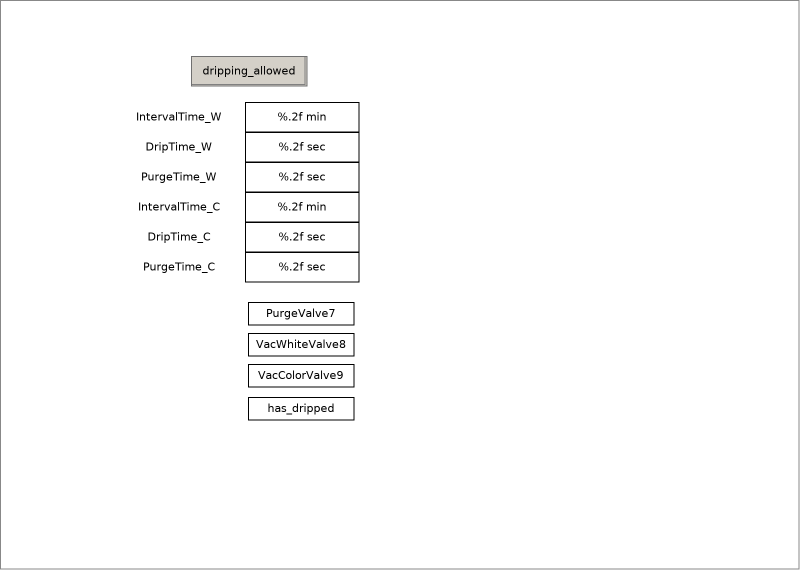
VISUALIZATION VIS_Drip_purge  // 800x570
    Button (191,56 116x30), "dripping_allowed", colour toggle: GVL_API.stMU.dripping_allowed
        toggle GVL_API.stMU.dripping_allowed
    RoundedRectangle (248,302 106x23), "PurgeValve7", colour toggle: P_MaintenanceUnit.FB_drip_purge.PurgeValve7
    Label (122,102 114x30), "IntervalTime_W"
    Label (122,132 114x30), "DripTime_W"
    Label (122,222 114x30), "DripTime_C"
    Label (122,162 114x30), "PurgeTime_W"
    Label (122,192 114x30), "IntervalTime_C"
    Label (122,252 114x30), "PurgeTime_C"
    Rectangle (245,102 114x30), "%.2f min", text variable: GVL_API.stMU.IntervalTime_W
        OnMouseDown: write GVL_API.stMU.IntervalTime_W via Default
    Rectangle (245,132 114x30), "%.2f sec", text variable: GVL_API.stMU.DripTime_W
        OnMouseDown: write GVL_API.stMU.DripTime_W via Default
    Rectangle (245,162 114x30), "%.2f sec", text variable: GVL_API.stMU.PurgeTime_W
        OnMouseDown: write GVL_API.stMU.PurgeTime_W via Default
    Rectangle (245,192 114x30), "%.2f min", text variable: GVL_API.stMU.IntervalTime_C
        OnMouseDown: write GVL_API.stMU.IntervalTime_C via Default
    Rectangle (245,222 114x30), "%.2f sec", text variable: GVL_API.stMU.DripTime_C
        OnMouseDown: write GVL_API.stMU.DripTime_C via Default
    Rectangle (245,252 114x30), "%.2f sec", text variable: GVL_API.stMU.PurgeTime_C
        OnMouseDown: write GVL_API.stMU.PurgeTime_C via Default
    RoundedRectangle (248,333 106x23), "VacWhiteValve8", colour toggle: P_MaintenanceUnit.FB_drip_purge.VacWhiteValve8
    RoundedRectangle (248,364 106x23), "VacColorValve9", colour toggle: P_MaintenanceUnit.FB_drip_purge.VacColorValve9
    RoundedRectangle (248,397 106x23), "has_dripped", colour toggle: GVL_API.stMU.has_dripped
END_VISUALIZATION

(* stored: Version 1.1.0.1, ProductVersion 3.1.4024.11
   Visu VIS_Drip_purge: Id {697ce32a-f504-481e-bcdb-767aa358c5cf} *)
